(*********************************** G.D S.p.A. - Technical Department ***********************************
============= PROGRAM INFO ============
FOLDER:             TBD
MACHINES INVOLVED:  TBD 

============= DESCRIPTION =============
csp main program

============= REVISIONS ===============
Date		Version	 	Author      	Description             
----------	-------		------------  	--------------------------------------------
2019/04/05 	0000.00	 	M.Grasso		Creation of the PRG

**********************************************************************************************************)
(*$R
	process_ref := prc;
$*)
PROGRAM csp_case_main
VAR
	prc:												process;
	prc_path:											STRING;
END_VAR


VAR_OUTPUT
	o_reset_button:										BOOL;
	o_start_button:										BOOL;
END_VAR

_read_var_input();

_object_manager();

IF NOT objects_running()
THEN
	RETURN;	
END_IF

_read_process_image();

_mode_manager();

CASE process_get_mode(prc) of
	MODE_ABSENT,
	MODE_INACTIVE:
		RETURN;
	MODE_TEST:
		_handle_process_test();
END_CASE

_set_runtime_properties();

(********************************* BODY *********************************)

(************************************************************************)

_handle_messages();

_write_output();

ACTION _handle_messages:
;
END_ACTION

ACTION _handle_process_test:
;
END_ACTION

ACTION _mode_manager:
IF process_mode_req_is_pending(prc)
THEN
    process_apply_mode_req_first_step(prc);
    CASE process_get_mode(prc) OF
        MODE_TO_ABSENT:
			;
        MODE_TO_INACTIVE:
			;
        MODE_TO_TEST:
			;
        MODE_TO_OPERATIONAL:
			;
    END_CASE
    process_apply_mode_req_second_step(prc);
END_IF
END_ACTION

ACTION _object_manager:
IF objects_initialization()
THEN
	sub_process_init(
		object_name					:= 'csp_case_main.prc', 
		process						:= csp_case.prc, 
		CONVERSION_this				:= prc);
		
	prc_path 						:= process_get_path(prc);
END_IF

IF objects_running()
THEN
	process_cycle(prc);
END_IF
END_ACTION

ACTION _read_process_image:
;
END_ACTION

ACTION _read_var_input:

END_ACTION

ACTION _set_runtime_properties:
;
END_ACTION

ACTION _write_output:
o_reset_button	:= csp_case_main_services_pushbuttons.reset_pressed;
o_start_button	:= csp_case_main_services_pushbuttons.start_pressed;
END_ACTION

END_PROGRAM

(* stored: Version 1.1.0.1, ProductVersion 3.1.4024.3
   POU csp_case_main: Id {67f35fcb-9b67-44aa-89a8-506d3495ea51}, SpecialFunc None
   Action _handle_messages: Id {a4a39ced-61e6-4b02-a9db-7ad1bec9730f}
   Action _handle_process_test: Id {9354002e-b4ba-42a9-a7c2-4f88c80aee33}
   Action _mode_manager: Id {4aaa66ae-1796-4b4f-be35-89597265f902}
   Action _object_manager: Id {144facca-a8d0-4679-baea-a36bbb347411}
   Action _read_process_image: Id {0e319b7a-23c3-4b97-8314-133793955825}
   Action _read_var_input: Id {33dc24b8-8dfa-4b5a-a193-03827c879fe3}
   Action _set_runtime_properties: Id {7f32af36-ba29-4dfd-a82d-db42b625982a}
   Action _write_output: Id {a204cf8c-7d90-40c2-b706-408742634f53} *)
